FUNCTION_BLOCK HeartBeat (* Composite Function Block Type *)
  (* Standard: 61499-2 *)
  (* Version 0.0, 25/02/2022, SESA197029, template *)
  PACKAGE SE.Nereda;
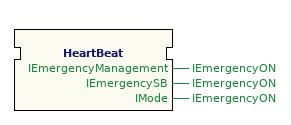
  PLUGS
    IEmergencyManagement : IEmergencyON;
    IEmergencySB : IEmergencyON;
    IMode : IEmergencyON;
  END_PLUGS
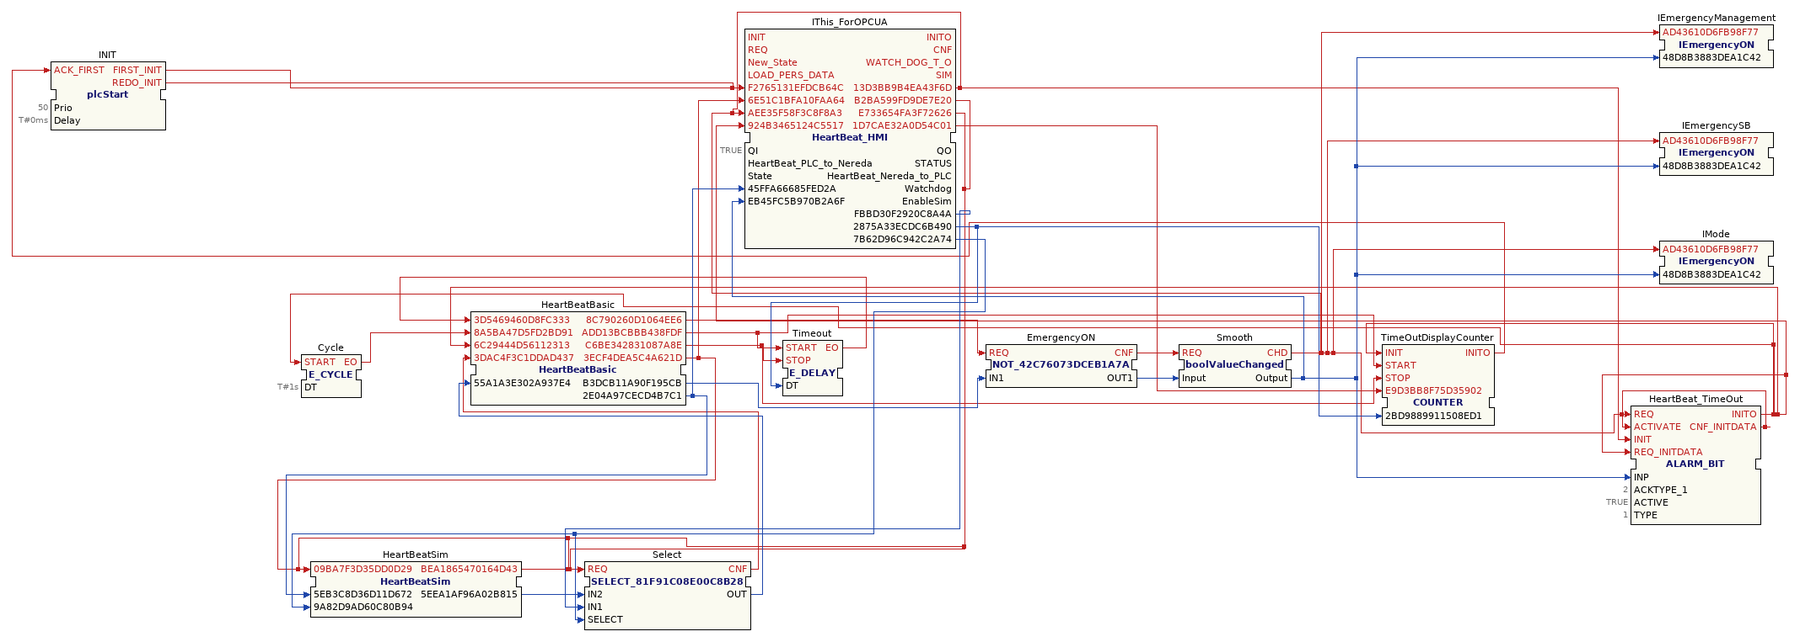
  (* 01 - FUNCTIONNAL INPUT INTERFACE *)
  (* 00 - INITIALIZATION *)
  (* 05 - LOGIC *)
  (* HEART BEAT SIMULATION *)
  (* 02 - FUNCTIONNAL OUTPUT INTERFACE *)
  (* 06 - HMI INTERFACE *)
  (* 07- REACTOR ALARM *)
  FBS
    IThis_ForOPCUA : HeartBeat_HMI(QI := TRUE);
    INIT : plcStart(Prio := 50, Delay := T#0ms);
    HeartBeatBasic : HeartBeatBasic;
    Cycle : E_CYCLE(DT := T#1s);
    EmergencyON : NOT_42C76073DCEB1A7A; {SET_ATTRIBUTE(Configuration.GenericFBType.InterfaceParams, Runtime.Standard#CNT:=1;OUT${CNT$}:BOOL)}
    Smooth : boolValueChanged;
    HeartBeat_TimeOut : ALARM_BIT(ACKTYPE_1 := 2, ACTIVE := TRUE, TYPE := 1);
    HeartBeatSim : HeartBeatSim;
    Select : SELECT_81F91C08E00C8B28; {SET_ATTRIBUTE(Configuration.GenericFBType.InterfaceParams, Runtime.Standard#CNT:=2;SELECT:BOOL;IN${CNT$}:BOOL)}
    Timeout : E_DELAY;
    TimeOutDisplayCounter : COUNTER; {SET_ATTRIBUTE(Configuration.Component.HideUnusedPorts, )}
  END_FBS
  EVENT_CONNECTIONS
    Timeout.EO TO HeartBeatBasic.3D5469460D8FC333;
    Cycle.EO TO HeartBeatBasic.8A5BA47D5FD2BD91;
    EmergencyON.CNF TO Smooth.REQ;
    Smooth.CHD TO IEmergencyManagement.AD43610D6FB98F77;
    Smooth.CHD TO IEmergencySB.AD43610D6FB98F77;
    Smooth.CHD TO IMode.AD43610D6FB98F77;
    HeartBeat_TimeOut.INITO TO TimeOutDisplayCounter.INIT;
    HeartBeat_TimeOut.INITO TO HeartBeatBasic.6C29444D56112313;
    HeartBeat_TimeOut.INITO TO Cycle.START;
    HeartBeatBasic.8C790260D1064EE6 TO EmergencyON.REQ;
    HeartBeatBasic.ADD13BCBBB438FDF TO Timeout.START;
    HeartBeatBasic.C6BE342831087A8E TO Timeout.STOP;
    HeartBeat_TimeOut.CNF_INITDATA TO HeartBeat_TimeOut.REQ;
    HeartBeat_TimeOut.CNF_INITDATA TO HeartBeat_TimeOut.ACTIVATE;
    IThis_ForOPCUA.13D3BB9B4EA43F6D TO HeartBeat_TimeOut.INIT;
    HeartBeat_TimeOut.INITO TO HeartBeat_TimeOut.REQ_INITDATA;
    HeartBeatBasic.3ECF4DEA5C4A621D TO HeartBeatSim.09BA7F3D35DD0D29;
    HeartBeatSim.BEA1865470164D43 TO Select.REQ;
    Select.CNF TO HeartBeatBasic.3DAC4F3C1DDAD437;
    INIT.FIRST_INIT TO IThis_ForOPCUA.F2765131EFDCB64C;
    INIT.REDO_INIT TO IThis_ForOPCUA.F2765131EFDCB64C;
    HeartBeatBasic.3ECF4DEA5C4A621D TO IThis_ForOPCUA.6E51C1BFA10FAA64;
    Smooth.CHD TO IThis_ForOPCUA.AEE35F58F3C8F8A3;
    IThis_ForOPCUA.13D3BB9B4EA43F6D TO IThis_ForOPCUA.AEE35F58F3C8F8A3;
    IThis_ForOPCUA.B2BA599FD9DE7E20 TO Select.REQ;
    IThis_ForOPCUA.E733654FA3F72626 TO HeartBeatSim.09BA7F3D35DD0D29;
    IThis_ForOPCUA.E733654FA3F72626 TO Select.REQ;
    HeartBeat_TimeOut.INITO TO IThis_ForOPCUA.924B3465124C5517;
    Smooth.CHD TO HeartBeat_TimeOut.REQ;
    TimeOutDisplayCounter.INITO TO INIT.ACK_FIRST;
    HeartBeatBasic.ADD13BCBBB438FDF TO TimeOutDisplayCounter.START;
    HeartBeatBasic.C6BE342831087A8E TO TimeOutDisplayCounter.STOP;
    IThis_ForOPCUA.1D7CAE32A0D54C01 TO TimeOutDisplayCounter.E9D3BB8F75D35902;
  END_CONNECTIONS
  DATA_CONNECTIONS
    EmergencyON.OUT1 TO Smooth.Input;
    Smooth.Output TO IEmergencyManagement.48D8B3883DEA1C42;
    Smooth.Output TO IEmergencySB.48D8B3883DEA1C42;
    Smooth.Output TO IMode.48D8B3883DEA1C42;
    HeartBeatBasic.B3DCB11A90F195CB TO EmergencyON.IN1;
    HeartBeatBasic.2E04A97CECD4B7C1 TO HeartBeatSim.5EB3C8D36D11D672;
    HeartBeatSim.5EEA1AF96A02B815 TO Select.IN2;
    Select.OUT TO HeartBeatBasic.55A1A3E302A937E4;
    HeartBeatBasic.2E04A97CECD4B7C1 TO IThis_ForOPCUA.45FFA66685FED2A;
    Smooth.Output TO IThis_ForOPCUA.EB45FC5B970B2A6F;
    IThis_ForOPCUA.FBBD30F2920C8A4A TO Select.IN1;
    IThis_ForOPCUA.2875A33ECDC6B490 TO Timeout.DT;
    IThis_ForOPCUA.7B62D96C942C2A74 TO HeartBeatSim.9A82D9AD60C80B94;
    IThis_ForOPCUA.7B62D96C942C2A74 TO Select.SELECT;
    Smooth.Output TO HeartBeat_TimeOut.INP;
    IThis_ForOPCUA.2875A33ECDC6B490 TO TimeOutDisplayCounter.2BD9889911508ED1;
  END_CONNECTIONS
END_FUNCTION_BLOCK
